{attribute 'qualified_only'}
{attribute 'strict'}
{attribute 'to_string'}
TYPE eHeatPumpMode :
(
	Standby := 0,
	Cooling := 1,
	Heating := 2
)UINT := Standby;
END_TYPE

(* stored: Version 1.1.0.1, ProductVersion 3.1.4026.18
   DUT eHeatPumpMode: Id {ed18c51f-e452-49d9-933b-77537eb36aea} *)
